FUNCTION_BLOCK T_CommandQueue_ClearWithHighPriority_ReturnTrue EXTENDS T_UnitTestBase
VAR
  command : T_CommandTask;
  commandQueue : T_CommandQueue;
  myTestState, prevState : (ARRANGE, ACT, ASSERT);
  actual : UINT := 0;
  expected : UINT := 0;
END_VAR

CASE myTestState OF
  ARRANGE:
	commandQueue.AddHighPriority(command);
    myTestState := ACT;
  
  ACT:
    commandQueue.clear();
    actual := commandQueue.Count;
	myTestState := ASSERT;
	
  ASSERT:
  	
    assertion.AssertEquals_UINT(expected, actual, 'commandQueue.clear High Priority = TRUE');
    myTestState := ARRANGE;
    TestFinished();
END_CASE

END_FUNCTION_BLOCK

(* stored: Version 1.1.0.1, ProductVersion 3.1.4024.12
   POU T_CommandQueue_ClearWithHighPriority_ReturnTrue: Id {a84f7941-4657-4300-bac0-b6f2e65d9deb}, SpecialFunc None *)
